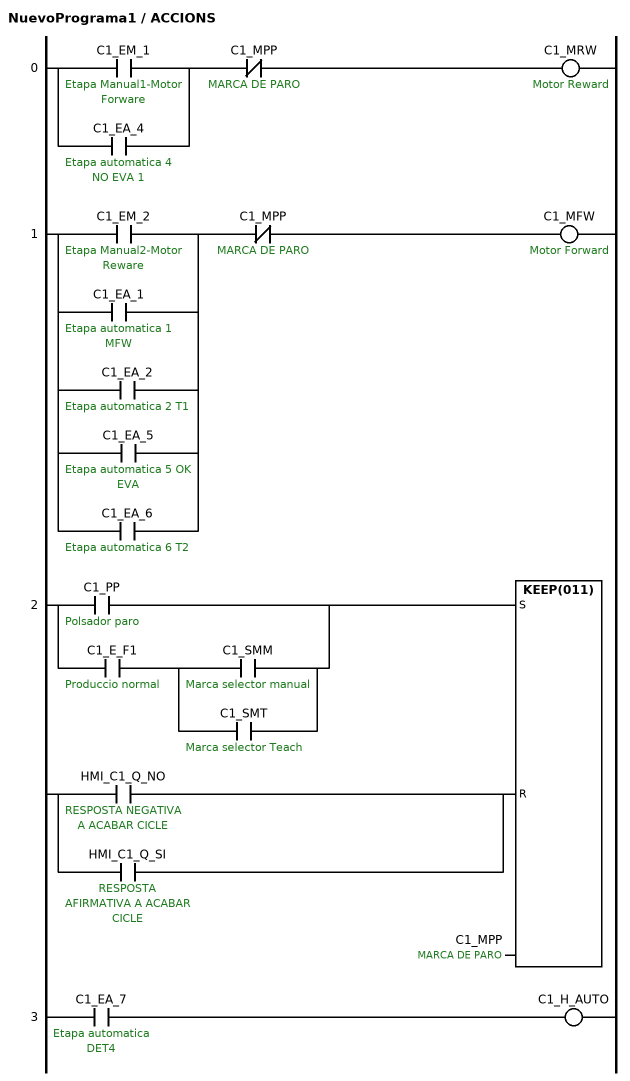
; [picture p24: NuevoPrograma1 / ACCIONS, rungs 0-3]
; rung 0
LD C1_EM_1  ; Etapa Manual1-Motor Forware
OR C1_EA_4  ; Etapa automatica 4 NO EVA 1
ANDNOT C1_MPP  ; MARCA DE PARO
OUT C1_MRW  ; Motor Reward
; rung 1
LD C1_EM_2  ; Etapa Manual2-Motor Reware
OR C1_EA_1  ; Etapa automatica 1 MFW
OR C1_EA_2  ; Etapa automatica 2 T1
OR C1_EA_5  ; Etapa automatica 5 OK EVA
OR C1_EA_6  ; Etapa automatica 6 T2
ANDNOT C1_MPP  ; MARCA DE PARO
OUT C1_MFW  ; Motor Forward
; rung 2
LD C1_PP  ; Polsador paro
LD C1_E_F1  ; Produccio normal
LD C1_SMM  ; Marca selector manual
OR C1_SMT  ; Marca selector Teach
ANDLD
ORLD
LD HMI_C1_Q_NO  ; RESPOSTA NEGATIVA A ACABAR CICLE
OR HMI_C1_Q_SI  ; RESPOSTA AFIRMATIVA A ACABAR CICLE
KEEP(011) C1_MPP  ; MARCA DE PARO
; rung 3
LD C1_EA_7  ; Etapa automatica DET4
OUT C1_H_AUTO

### Section ACCIONS_HMI

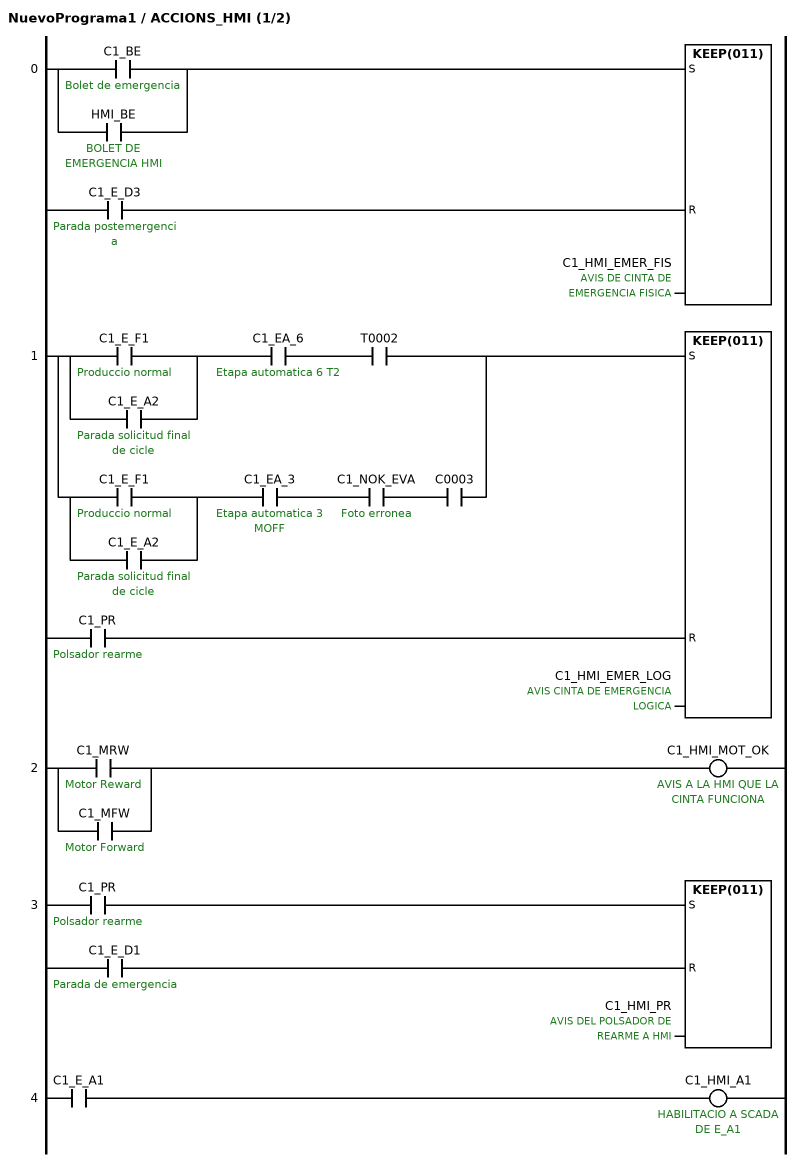
; rung 0
LD C1_BE  ; Bolet de emergencia
OR HMI_BE  ; BOLET DE EMERGENCIA HMI
LD C1_E_D3  ; Parada postemergencia
KEEP(011) C1_HMI_EMER_FIS  ; AVIS DE CINTA DE EMERGENCIA FISICA
; rung 1
LD C1_E_F1  ; Produccio normal
OR C1_E_A2  ; Parada solicitud final de cicle
AND C1_EA_6  ; Etapa automatica 6 T2
AND T0002
LD C1_E_F1  ; Produccio normal
OR C1_E_A2  ; Parada solicitud final de cicle
AND C1_EA_3  ; Etapa automatica 3 MOFF
AND C1_NOK_EVA  ; Foto erronea
AND C0003
ORLD
LD C1_PR  ; Polsador rearme
KEEP(011) C1_HMI_EMER_LOG  ; AVIS CINTA DE EMERGENCIA LOGICA
; rung 2
LD C1_MRW  ; Motor Reward
OR C1_MFW  ; Motor Forward
OUT C1_HMI_MOT_OK  ; AVIS A LA HMI QUE LA CINTA FUNCIONA
; rung 3
LD C1_PR  ; Polsador rearme
LD C1_E_D1  ; Parada de emergencia
KEEP(011) C1_HMI_PR  ; AVIS DEL POLSADOR DE REARME A HMI
; rung 4
LD C1_E_A1
OUT C1_HMI_A1  ; HABILITACIO A SCADA DE E_A1

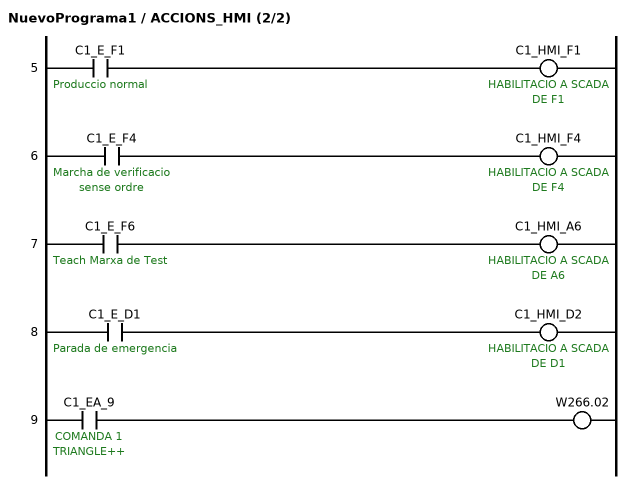
; rung 5
LD C1_E_F1  ; Produccio normal
OUT C1_HMI_F1  ; HABILITACIO A SCADA DE F1
; rung 6
LD C1_E_F4  ; Marcha de verificacio sense ordre
OUT C1_HMI_F4  ; HABILITACIO A SCADA DE F4
; rung 7
LD C1_E_F6  ; Teach Marxa de Test
OUT C1_HMI_A6  ; HABILITACIO A SCADA DE A6
; rung 8
LD C1_E_D1  ; Parada de emergencia
OUT C1_HMI_D2  ; HABILITACIO A SCADA DE D1
; rung 9
LD C1_EA_9  ; COMANDA 1 TRIANGLE++
OUT W266.02

### Section ACCIONS_ROBOT

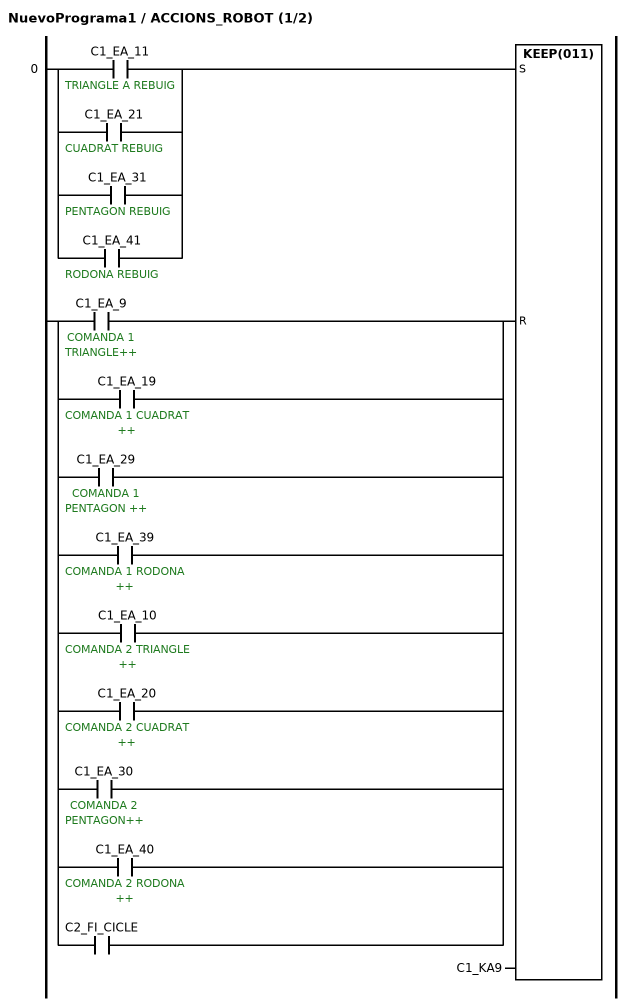
; rung 0
LD C1_EA_11  ; TRIANGLE A REBUIG
OR C1_EA_21  ; CUADRAT REBUIG
OR C1_EA_31  ; PENTAGON REBUIG
OR C1_EA_41  ; RODONA REBUIG
LD C1_EA_9  ; COMANDA 1 TRIANGLE++
OR C1_EA_19  ; COMANDA 1 CUADRAT ++
OR C1_EA_29  ; COMANDA 1 PENTAGON ++
OR C1_EA_39  ; COMANDA 1 RODONA ++
OR C1_EA_10  ; COMANDA 2 TRIANGLE ++
OR C1_EA_20  ; COMANDA 2 CUADRAT ++
OR C1_EA_30  ; COMANDA 2 PENTAGON++
OR C1_EA_40  ; COMANDA 2 RODONA ++
OR C2_FI_CICLE
KEEP(011) C1_KA9

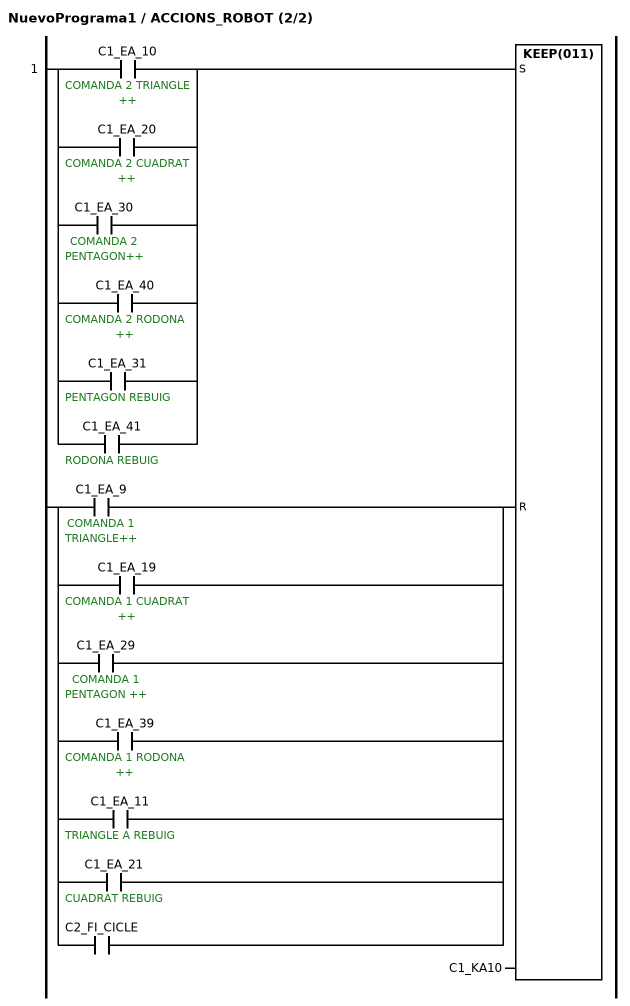
; rung 1
LD C1_EA_10  ; COMANDA 2 TRIANGLE ++
OR C1_EA_20  ; COMANDA 2 CUADRAT ++
OR C1_EA_30  ; COMANDA 2 PENTAGON++
OR C1_EA_40  ; COMANDA 2 RODONA ++
OR C1_EA_31  ; PENTAGON REBUIG
OR C1_EA_41  ; RODONA REBUIG
LD C1_EA_9  ; COMANDA 1 TRIANGLE++
OR C1_EA_19  ; COMANDA 1 CUADRAT ++
OR C1_EA_29  ; COMANDA 1 PENTAGON ++
OR C1_EA_39  ; COMANDA 1 RODONA ++
OR C1_EA_11  ; TRIANGLE A REBUIG
OR C1_EA_21  ; CUADRAT REBUIG
OR C2_FI_CICLE
KEEP(011) C1_KA10

### Section ACCIONS_CT2

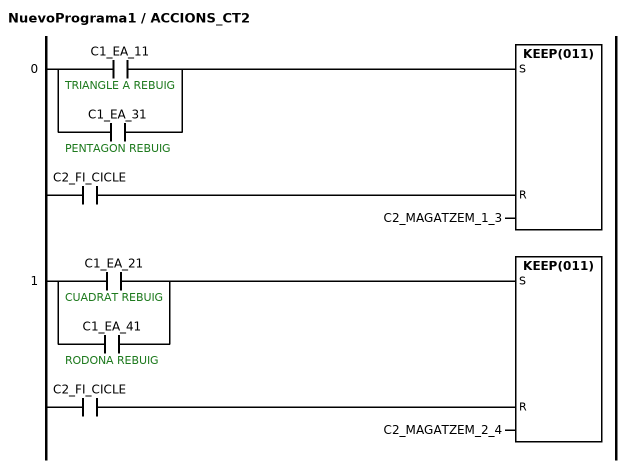
; rung 0
LD C1_EA_11  ; TRIANGLE A REBUIG
OR C1_EA_31  ; PENTAGON REBUIG
LD C2_FI_CICLE
KEEP(011) C2_MAGATZEM_1_3
; rung 1
LD C1_EA_21  ; CUADRAT REBUIG
OR C1_EA_41  ; RODONA REBUIG
LD C2_FI_CICLE
KEEP(011) C2_MAGATZEM_2_4

### Section END
; rung 0
END(001)